(* Logix 5000 project; controller SX_V040001_C001 vendor 1 type 14 code 77 rev 16.23; software revision 16.04; part 19 of 35 *)
(* tags used below, declared in another part *)
   ALARM_BITS : INT[10];
   ALARM_BUFFER : INT[10];
   ALL_KINDS : INT[90];
   Basic : INT;
   CMD : INT[36];
   DRIVE : INT[32];
   DRIVE_INTERVAL : INT[8];
   EMPTYING : INT[18];
   G_DInput : DINT[3];
   G_DOutput : DINT[3];
   loading : INT[19];
   m_alarm_exist : BOOL;
   m_on_off_line : BOOL;
   m_power_up : BOOL;
   M_SIMU_ON_OFF : BOOL;
   MESSAGE_BITS : INT[8];
   METERING : INT[44];
   mw_minor_fault : DINT;
   NOTDOS : INT[6];
   PARAMETER : INT[501];
   pointer_alarm_buffer : DINT;
   pointer_bit_nr : DINT;
   pointer_word_nr : DINT;
   STATUS_GENERAL : INT[135];
(* MainProgram, continued *)

ROUTINE MainDriveInterval   (* ladder *)
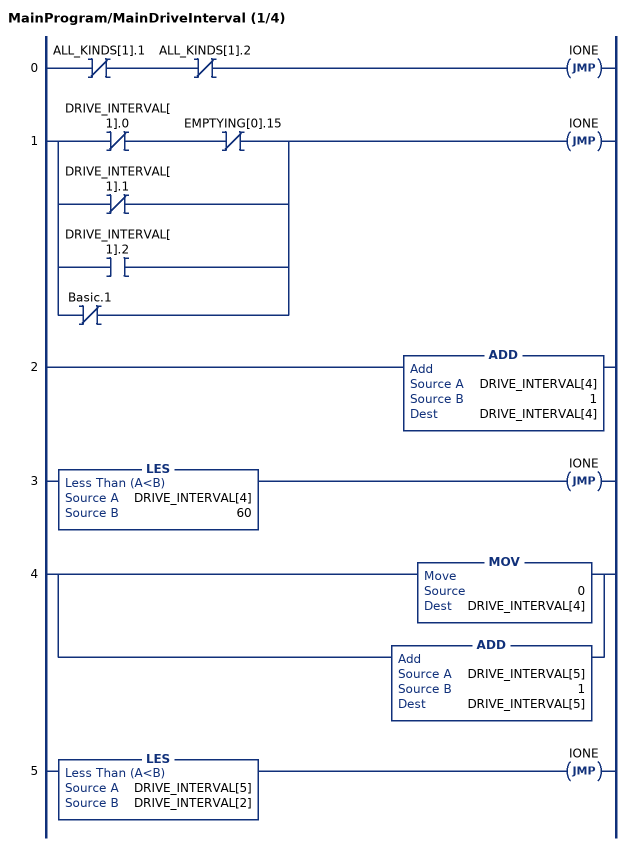
   0: XIO(ALL_KINDS[1].1)XIO(ALL_KINDS[1].2)JMP(IONE);
   1: [XIO(DRIVE_INTERVAL[1].0) XIO(EMPTYING[0].15) ,XIO(DRIVE_INTERVAL[1].1) ,XIC(DRIVE_INTERVAL[1].2) ,XIO(Basic.1) ]JMP(IONE);
   2: ADD(DRIVE_INTERVAL[4],1,DRIVE_INTERVAL[4]);
   3: LES(DRIVE_INTERVAL[4],60)JMP(IONE);
   4: [MOV(0,DRIVE_INTERVAL[4]) ,ADD(DRIVE_INTERVAL[5],1,DRIVE_INTERVAL[5]) ];
   5: LES(DRIVE_INTERVAL[5],DRIVE_INTERVAL[2])JMP(IONE);
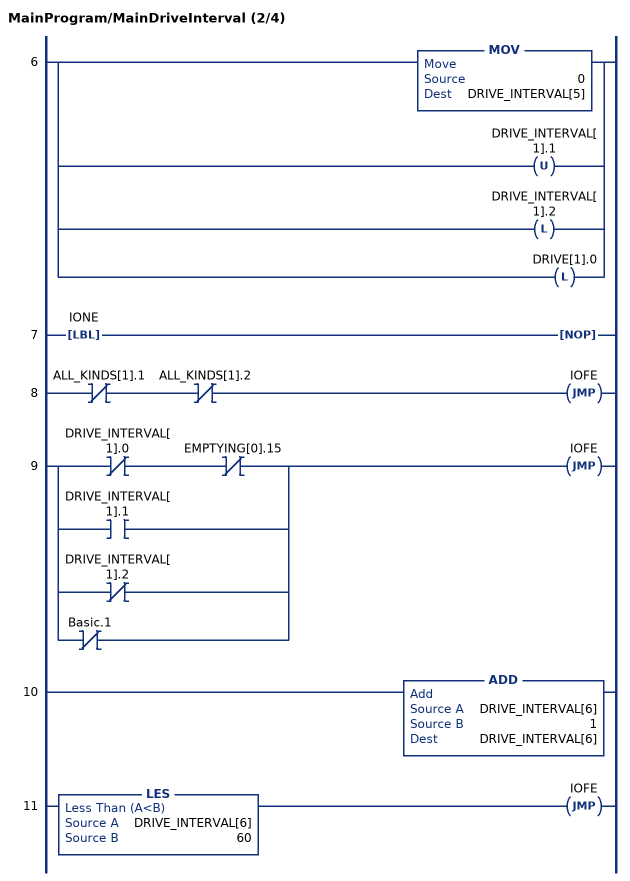
   6: [MOV(0,DRIVE_INTERVAL[5]) ,OTU(DRIVE_INTERVAL[1].1) ,OTL(DRIVE_INTERVAL[1].2) ,OTL(DRIVE[1].0) ];
   7: LBL(IONE)NOP();
   8: XIO(ALL_KINDS[1].1)XIO(ALL_KINDS[1].2)JMP(IOFE);
   9: [XIO(DRIVE_INTERVAL[1].0) XIO(EMPTYING[0].15) ,XIC(DRIVE_INTERVAL[1].1) ,XIO(DRIVE_INTERVAL[1].2) ,XIO(Basic.1) ]JMP(IOFE);
   10: ADD(DRIVE_INTERVAL[6],1,DRIVE_INTERVAL[6]);
   11: LES(DRIVE_INTERVAL[6],60)JMP(IOFE);
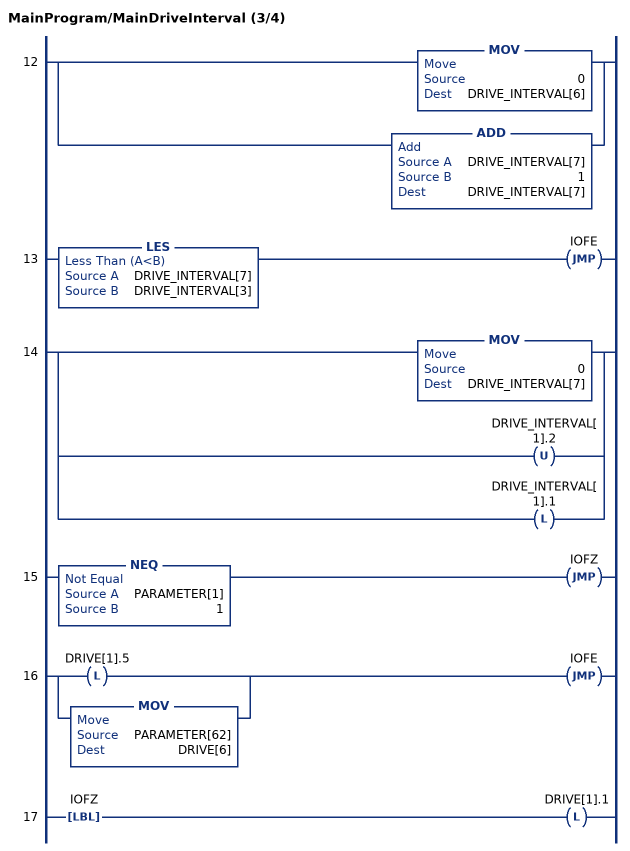
   12: [MOV(0,DRIVE_INTERVAL[6]) ,ADD(DRIVE_INTERVAL[7],1,DRIVE_INTERVAL[7]) ];
   13: LES(DRIVE_INTERVAL[7],DRIVE_INTERVAL[3])JMP(IOFE);
   14: [MOV(0,DRIVE_INTERVAL[7]) ,OTU(DRIVE_INTERVAL[1].2) ,OTL(DRIVE_INTERVAL[1].1) ];
   15: NEQ(PARAMETER[1],1)JMP(IOFZ);
   16: [OTL(DRIVE[1].5) ,MOV(PARAMETER[62],DRIVE[6]) ]JMP(IOFE);
   17: LBL(IOFZ)OTL(DRIVE[1].1);
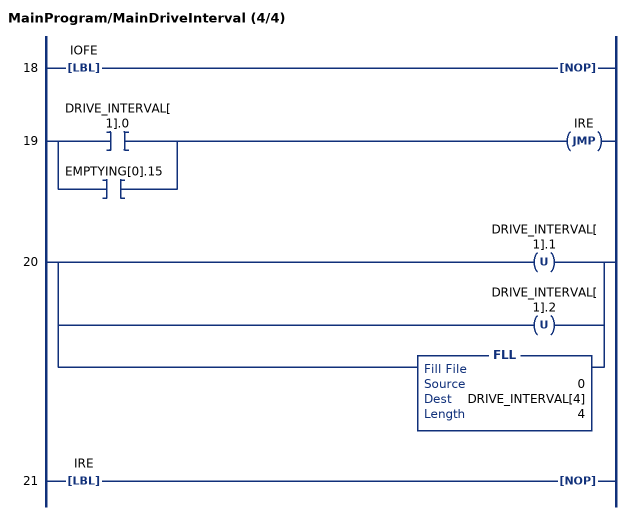
   18: LBL(IOFE)NOP();
   19: [XIC(DRIVE_INTERVAL[1].0) ,XIC(EMPTYING[0].15) ]JMP(IRE);
   20: [OTU(DRIVE_INTERVAL[1].1) ,OTU(DRIVE_INTERVAL[1].2) ,FLL(0,DRIVE_INTERVAL[4],4) ];
   21: LBL(IRE)NOP();
END_ROUTINE

ROUTINE MainRoutine   (* ladder *)
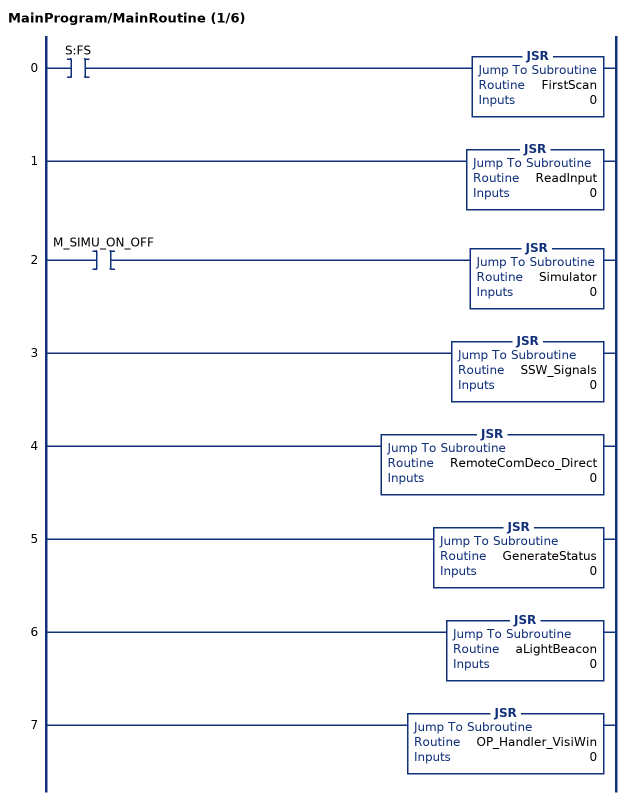
   0: XIC(S:FS)JSR(FirstScan,0);
   1: JSR(ReadInput,0);
   2: XIC(M_SIMU_ON_OFF)JSR(Simulator,0);
   3: JSR(SSW_Signals,0);
   4: JSR(RemoteComDeco_Direct,0);
   5: JSR(GenerateStatus,0);
   6: JSR(aLightBeacon,0);
   7: JSR(OP_Handler_VisiWin,0);
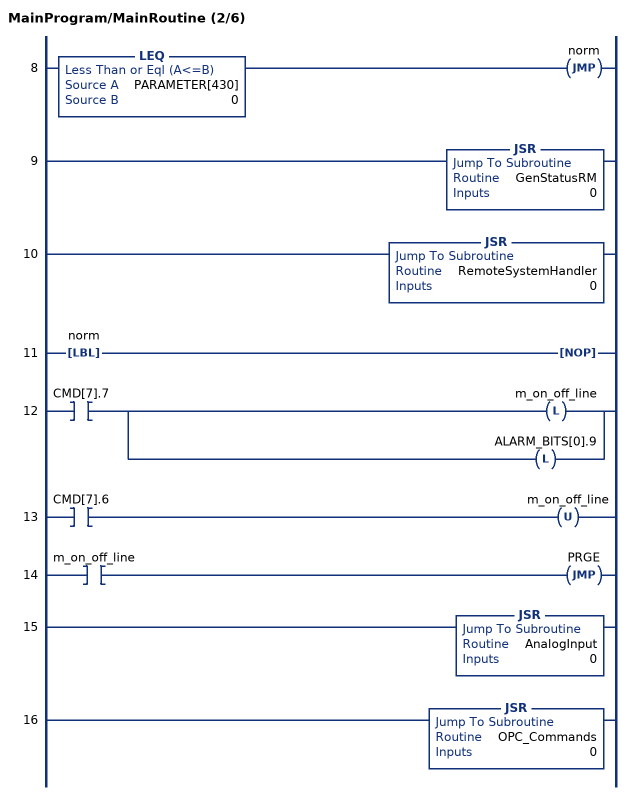
   8: LEQ(PARAMETER[430],0)JMP(norm);
   9: JSR(GenStatusRM,0);
   10: JSR(RemoteSystemHandler,0);
   11: LBL(norm)NOP();
   12: XIC(CMD[7].7)[OTL(m_on_off_line) ,OTL(ALARM_BITS[0].9) ];
   13: XIC(CMD[7].6)OTU(m_on_off_line);
   14: XIC(m_on_off_line)JMP(PRGE);
   15: JSR(AnalogInput,0);
   16: JSR(OPC_Commands,0);
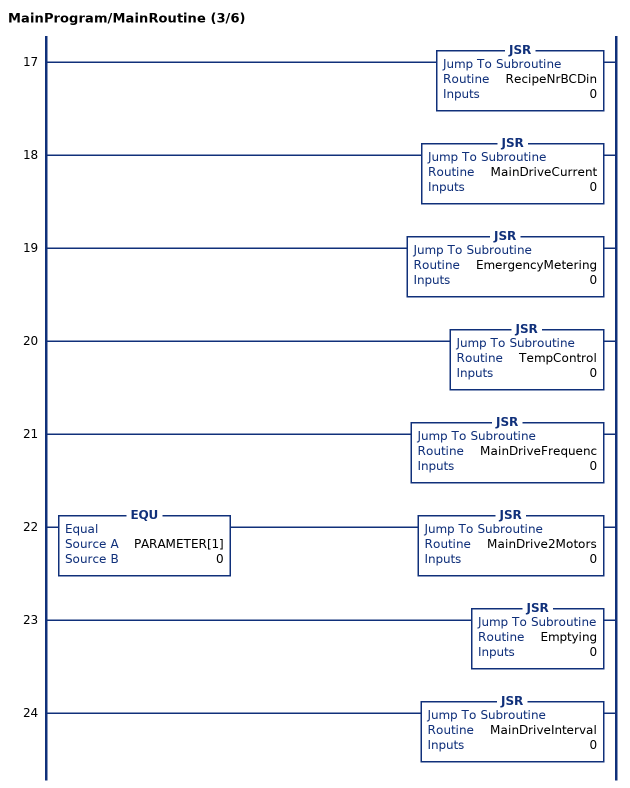
   17: JSR(RecipeNrBCDin,0);
   18: JSR(MainDriveCurrent,0);
   19: JSR(EmergencyMetering,0);
   20: JSR(TempControl,0);
   21: JSR(MainDriveFrequenc,0);
   22: EQU(PARAMETER[1],0)JSR(MainDrive2Motors,0);
   23: JSR(Emptying,0);
   24: JSR(MainDriveInterval,0);
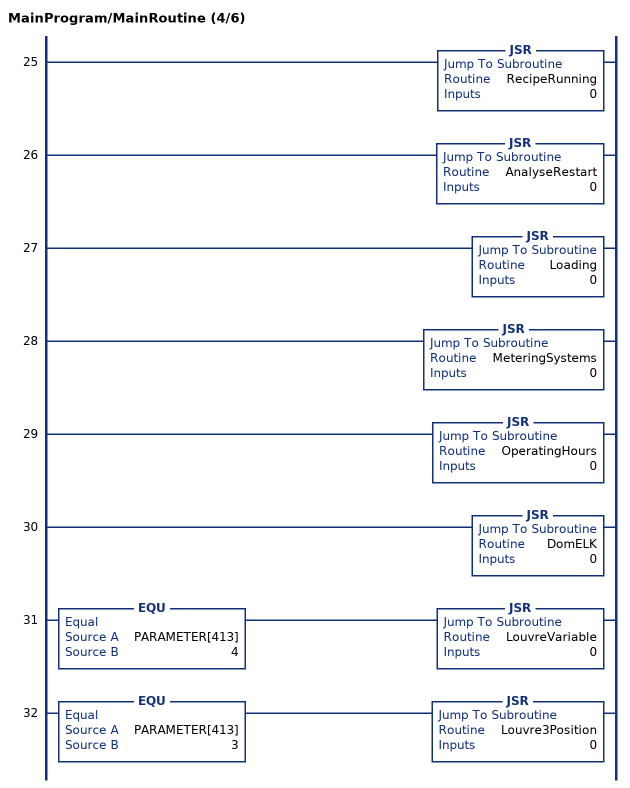
   25: JSR(RecipeRunning,0);
   26: JSR(AnalyseRestart,0);
   27: JSR(Loading,0);
   28: JSR(MeteringSystems,0);
   29: JSR(OperatingHours,0);
   30: JSR(DomELK,0);
   31: EQU(PARAMETER[413],4)JSR(LouvreVariable,0);
   32: EQU(PARAMETER[413],3)JSR(Louvre3Position,0);
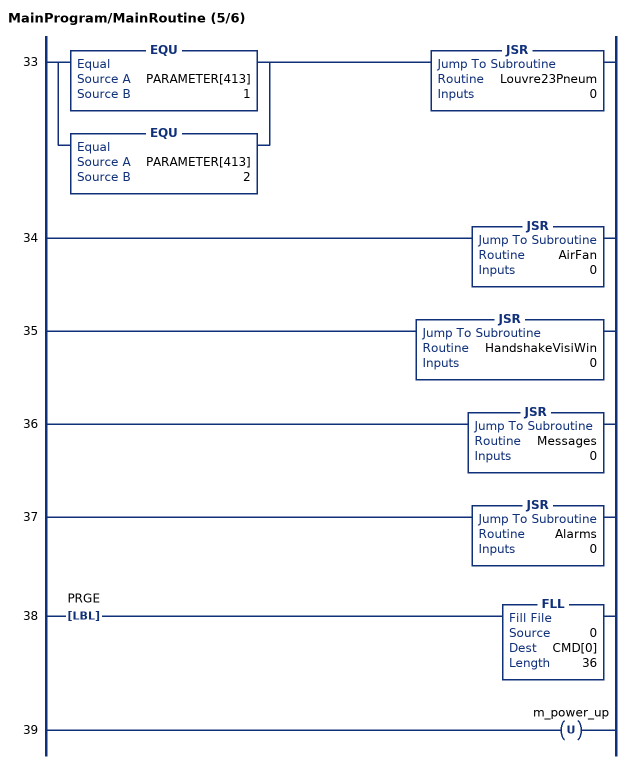
   33: [EQU(PARAMETER[413],1) ,EQU(PARAMETER[413],2) ]JSR(Louvre23Pneum,0);
   34: JSR(AirFan,0);
   35: JSR(HandshakeVisiWin,0);
   36: JSR(Messages,0);
   37: JSR(Alarms,0);
   38: LBL(PRGE)FLL(0,CMD[0],36);
   39: OTU(m_power_up);
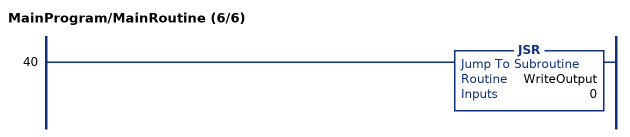
   40: JSR(WriteOutput,0);
END_ROUTINE

ROUTINE MessageBitToNumber   (* ladder *)
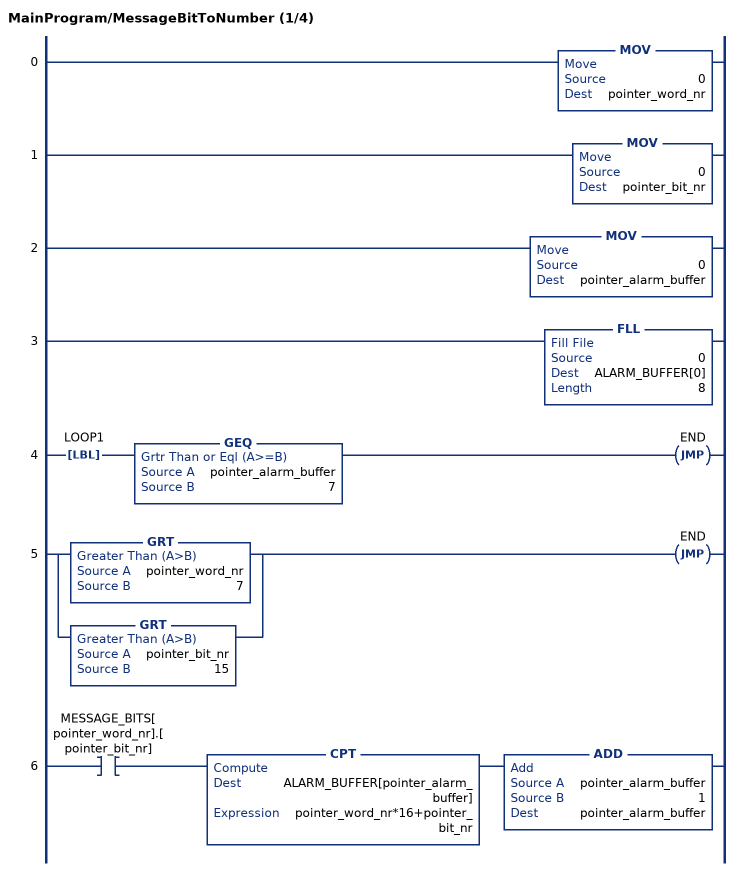
   0: MOV(0,pointer_word_nr);
   1: MOV(0,pointer_bit_nr);
   2: MOV(0,pointer_alarm_buffer);
   3: FLL(0,ALARM_BUFFER[0],8);
   4: LBL(LOOP1)GEQ(pointer_alarm_buffer,7)JMP(END);
   5: [GRT(pointer_word_nr,7) ,GRT(pointer_bit_nr,15) ]JMP(END);
   6: XIC(MESSAGE_BITS[pointer_word_nr].[pointer_bit_nr])CPT(ALARM_BUFFER[pointer_alarm_buffer],pointer_word_nr*16+pointer_bit_nr)ADD(pointer_alarm_buffer,1,pointer_alarm_buffer);
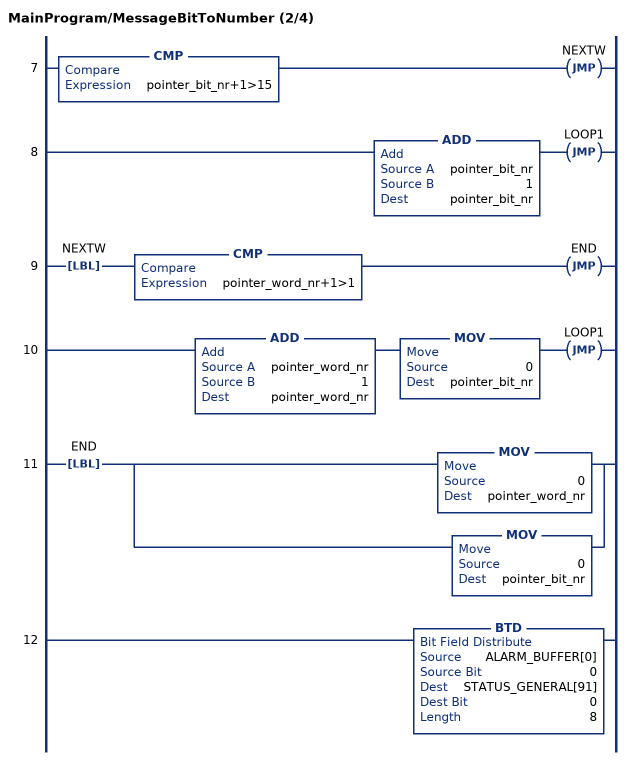
   7: CMP(pointer_bit_nr+1>15)JMP(NEXTW);
   8: ADD(pointer_bit_nr,1,pointer_bit_nr)JMP(LOOP1);
   9: LBL(NEXTW)CMP(pointer_word_nr+1>1)JMP(END);
   10: ADD(pointer_word_nr,1,pointer_word_nr)MOV(0,pointer_bit_nr)JMP(LOOP1);
   11: LBL(END)[MOV(0,pointer_word_nr) ,MOV(0,pointer_bit_nr) ];
   12: BTD(ALARM_BUFFER[0],0,STATUS_GENERAL[91],0,8);
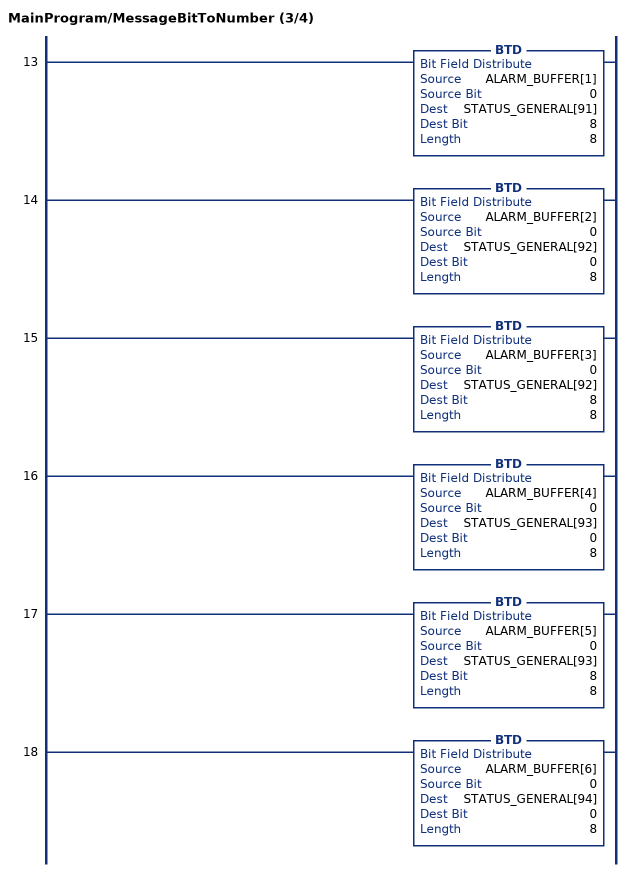
   13: BTD(ALARM_BUFFER[1],0,STATUS_GENERAL[91],8,8);
   14: BTD(ALARM_BUFFER[2],0,STATUS_GENERAL[92],0,8);
   15: BTD(ALARM_BUFFER[3],0,STATUS_GENERAL[92],8,8);
   16: BTD(ALARM_BUFFER[4],0,STATUS_GENERAL[93],0,8);
   17: BTD(ALARM_BUFFER[5],0,STATUS_GENERAL[93],8,8);
   18: BTD(ALARM_BUFFER[6],0,STATUS_GENERAL[94],0,8);
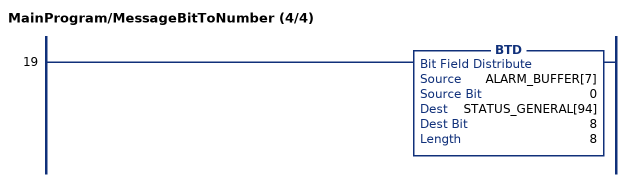
   19: BTD(ALARM_BUFFER[7],0,STATUS_GENERAL[94],8,8);
END_ROUTINE

ROUTINE Messages   (* ladder *)
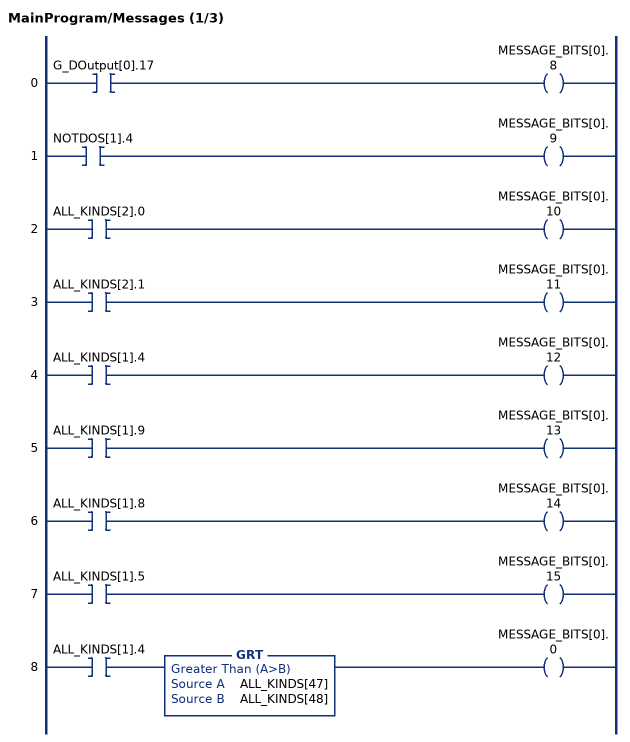
   0: XIC(G_DOutput[0].17)OTE(MESSAGE_BITS[0].8);
   1: XIC(NOTDOS[1].4)OTE(MESSAGE_BITS[0].9);
   2: XIC(ALL_KINDS[2].0)OTE(MESSAGE_BITS[0].10);
   3: XIC(ALL_KINDS[2].1)OTE(MESSAGE_BITS[0].11);
   4: XIC(ALL_KINDS[1].4)OTE(MESSAGE_BITS[0].12);
   5: XIC(ALL_KINDS[1].9)OTE(MESSAGE_BITS[0].13);
   6: XIC(ALL_KINDS[1].8)OTE(MESSAGE_BITS[0].14);
   7: XIC(ALL_KINDS[1].5)OTE(MESSAGE_BITS[0].15);
   8: XIC(ALL_KINDS[1].4)GRT(ALL_KINDS[47],ALL_KINDS[48])OTE(MESSAGE_BITS[0].0);
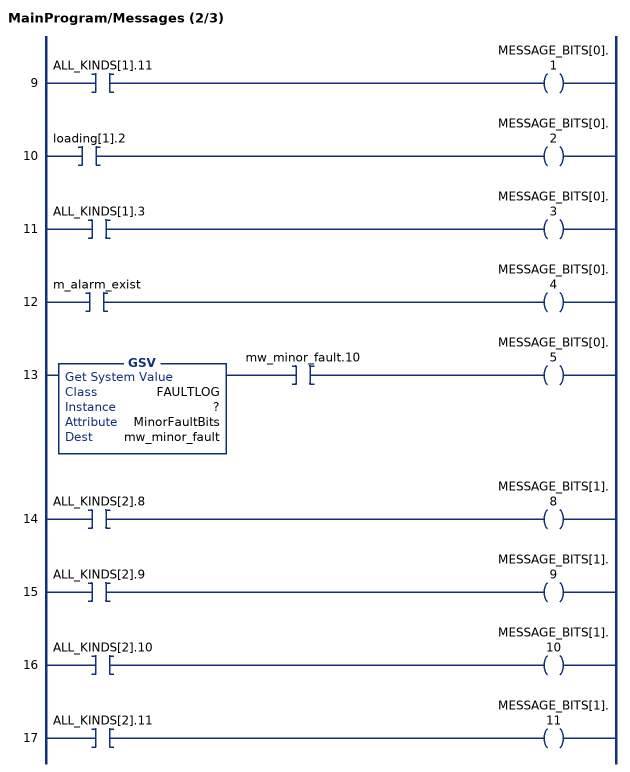
   9: XIC(ALL_KINDS[1].11)OTE(MESSAGE_BITS[0].1);
   10: XIC(loading[1].2)OTE(MESSAGE_BITS[0].2);
   11: XIC(ALL_KINDS[1].3)OTE(MESSAGE_BITS[0].3);
   12: XIC(m_alarm_exist)OTE(MESSAGE_BITS[0].4);
   13: GSV(FAULTLOG,?,MinorFaultBits,mw_minor_fault)XIC(mw_minor_fault.10)OTE(MESSAGE_BITS[0].5);
   14: XIC(ALL_KINDS[2].8)OTE(MESSAGE_BITS[1].8);
   15: XIC(ALL_KINDS[2].9)OTE(MESSAGE_BITS[1].9);
   16: XIC(ALL_KINDS[2].10)OTE(MESSAGE_BITS[1].10);
   17: XIC(ALL_KINDS[2].11)OTE(MESSAGE_BITS[1].11);
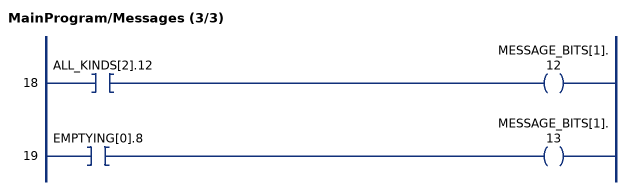
   18: XIC(ALL_KINDS[2].12)OTE(MESSAGE_BITS[1].12);
   19: XIC(EMPTYING[0].8)OTE(MESSAGE_BITS[1].13);
END_ROUTINE

ROUTINE MeteringSystems   (* ladder *)
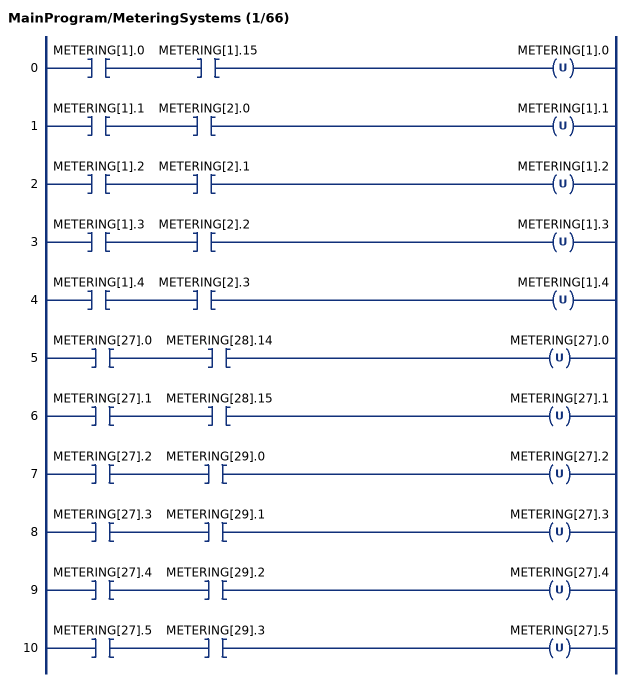
   0: XIC(METERING[1].0)XIC(METERING[1].15)OTU(METERING[1].0);
   1: XIC(METERING[1].1)XIC(METERING[2].0)OTU(METERING[1].1);
   2: XIC(METERING[1].2)XIC(METERING[2].1)OTU(METERING[1].2);
   3: XIC(METERING[1].3)XIC(METERING[2].2)OTU(METERING[1].3);
   4: XIC(METERING[1].4)XIC(METERING[2].3)OTU(METERING[1].4);
   5: XIC(METERING[27].0)XIC(METERING[28].14)OTU(METERING[27].0);
   6: XIC(METERING[27].1)XIC(METERING[28].15)OTU(METERING[27].1);
   7: XIC(METERING[27].2)XIC(METERING[29].0)OTU(METERING[27].2);
   8: XIC(METERING[27].3)XIC(METERING[29].1)OTU(METERING[27].3);
   9: XIC(METERING[27].4)XIC(METERING[29].2)OTU(METERING[27].4);
   10: XIC(METERING[27].5)XIC(METERING[29].3)OTU(METERING[27].5);
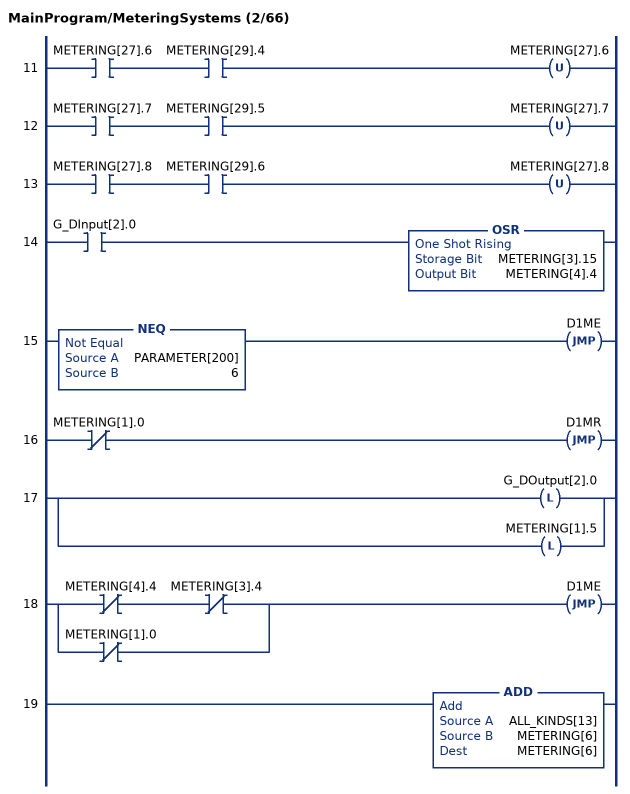
   11: XIC(METERING[27].6)XIC(METERING[29].4)OTU(METERING[27].6);
   12: XIC(METERING[27].7)XIC(METERING[29].5)OTU(METERING[27].7);
   13: XIC(METERING[27].8)XIC(METERING[29].6)OTU(METERING[27].8);
   14: XIC(G_DInput[2].0)OSR(METERING[3].15,METERING[4].4);
   15: NEQ(PARAMETER[200],6)JMP(D1ME);
   16: XIO(METERING[1].0)JMP(D1MR);
   17: [OTL(G_DOutput[2].0) ,OTL(METERING[1].5) ];
   18: [XIO(METERING[4].4) XIO(METERING[3].4) ,XIO(METERING[1].0) ]JMP(D1ME);
   19: ADD(ALL_KINDS[13],METERING[6],METERING[6]);
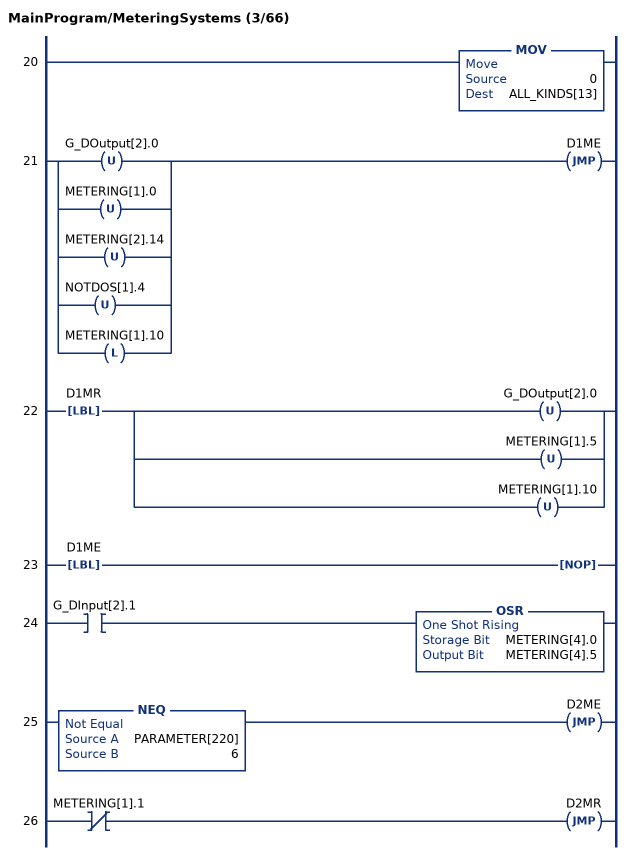
   20: MOV(0,ALL_KINDS[13]);
   21: [OTU(G_DOutput[2].0) ,OTU(METERING[1].0) ,OTU(METERING[2].14) ,OTU(NOTDOS[1].4) ,OTL(METERING[1].10) ]JMP(D1ME);
   22: LBL(D1MR)[OTU(G_DOutput[2].0) ,OTU(METERING[1].5) ,OTU(METERING[1].10) ];
   23: LBL(D1ME)NOP();
   24: XIC(G_DInput[2].1)OSR(METERING[4].0,METERING[4].5);
   25: NEQ(PARAMETER[220],6)JMP(D2ME);
   26: XIO(METERING[1].1)JMP(D2MR);
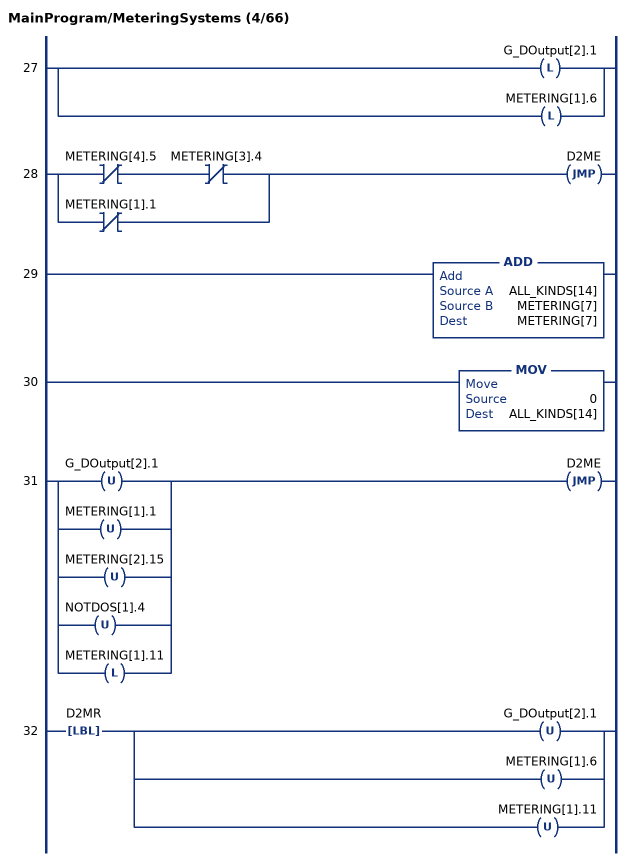
   27: [OTL(G_DOutput[2].1) ,OTL(METERING[1].6) ];
   28: [XIO(METERING[4].5) XIO(METERING[3].4) ,XIO(METERING[1].1) ]JMP(D2ME);
   29: ADD(ALL_KINDS[14],METERING[7],METERING[7]);
   30: MOV(0,ALL_KINDS[14]);
   31: [OTU(G_DOutput[2].1) ,OTU(METERING[1].1) ,OTU(METERING[2].15) ,OTU(NOTDOS[1].4) ,OTL(METERING[1].11) ]JMP(D2ME);
   32: LBL(D2MR)[OTU(G_DOutput[2].1) ,OTU(METERING[1].6) ,OTU(METERING[1].11) ];
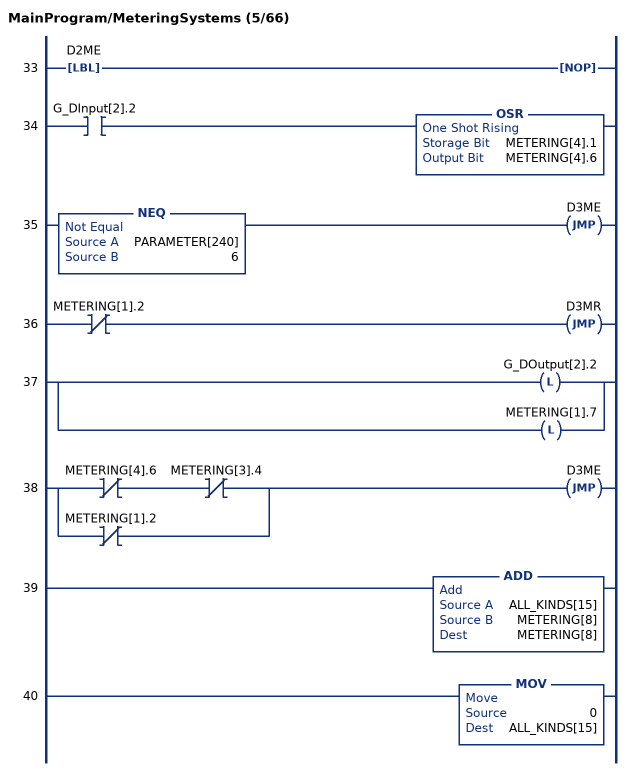
   33: LBL(D2ME)NOP();
   34: XIC(G_DInput[2].2)OSR(METERING[4].1,METERING[4].6);
   35: NEQ(PARAMETER[240],6)JMP(D3ME);
   36: XIO(METERING[1].2)JMP(D3MR);
   37: [OTL(G_DOutput[2].2) ,OTL(METERING[1].7) ];
   38: [XIO(METERING[4].6) XIO(METERING[3].4) ,XIO(METERING[1].2) ]JMP(D3ME);
   39: ADD(ALL_KINDS[15],METERING[8],METERING[8]);
   40: MOV(0,ALL_KINDS[15]);
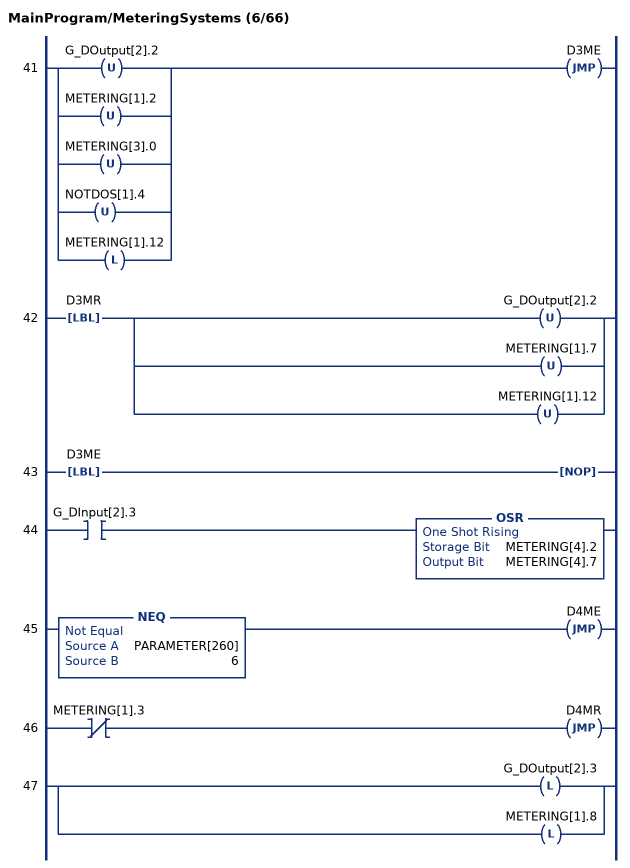
   41: [OTU(G_DOutput[2].2) ,OTU(METERING[1].2) ,OTU(METERING[3].0) ,OTU(NOTDOS[1].4) ,OTL(METERING[1].12) ]JMP(D3ME);
   42: LBL(D3MR)[OTU(G_DOutput[2].2) ,OTU(METERING[1].7) ,OTU(METERING[1].12) ];
   43: LBL(D3ME)NOP();
   44: XIC(G_DInput[2].3)OSR(METERING[4].2,METERING[4].7);
   45: NEQ(PARAMETER[260],6)JMP(D4ME);
   46: XIO(METERING[1].3)JMP(D4MR);
   47: [OTL(G_DOutput[2].3) ,OTL(METERING[1].8) ];
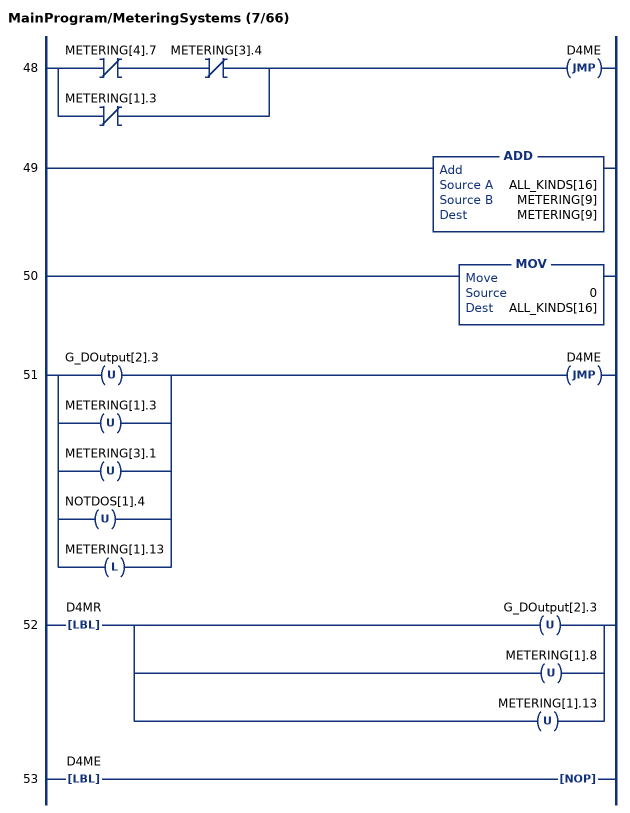
   48: [XIO(METERING[4].7) XIO(METERING[3].4) ,XIO(METERING[1].3) ]JMP(D4ME);
   49: ADD(ALL_KINDS[16],METERING[9],METERING[9]);
   50: MOV(0,ALL_KINDS[16]);
   51: [OTU(G_DOutput[2].3) ,OTU(METERING[1].3) ,OTU(METERING[3].1) ,OTU(NOTDOS[1].4) ,OTL(METERING[1].13) ]JMP(D4ME);
   52: LBL(D4MR)[OTU(G_DOutput[2].3) ,OTU(METERING[1].8) ,OTU(METERING[1].13) ];
   53: LBL(D4ME)NOP();
